FUNCTION_BLOCK FB_PRES_CNTRL
VAR_INPUT

END_VAR
VAR_IN_OUT
	Control : TYP_PRES_CNTRL_CONTROL;
	Parameter: TYP_PRES_CNTRL_PARAMETER;
END_VAR
VAR_OUTPUT
	Status : TYP_PRES_CNTRL_STATUS;
END_VAR
VAR
END_VAR

END_FUNCTION_BLOCK

(* stored: Version 1.1.0.1, ProductVersion 3.1.4024.12
   POU FB_PRES_CNTRL: Id {59080cdc-8ddf-4030-bdc0-c24b6df0f728}, SpecialFunc None *)
